// Mitsubishi GX Works2 project: 250627_단일공정순차제어(2)   PLC: Q02U

PROGRAM MAIN
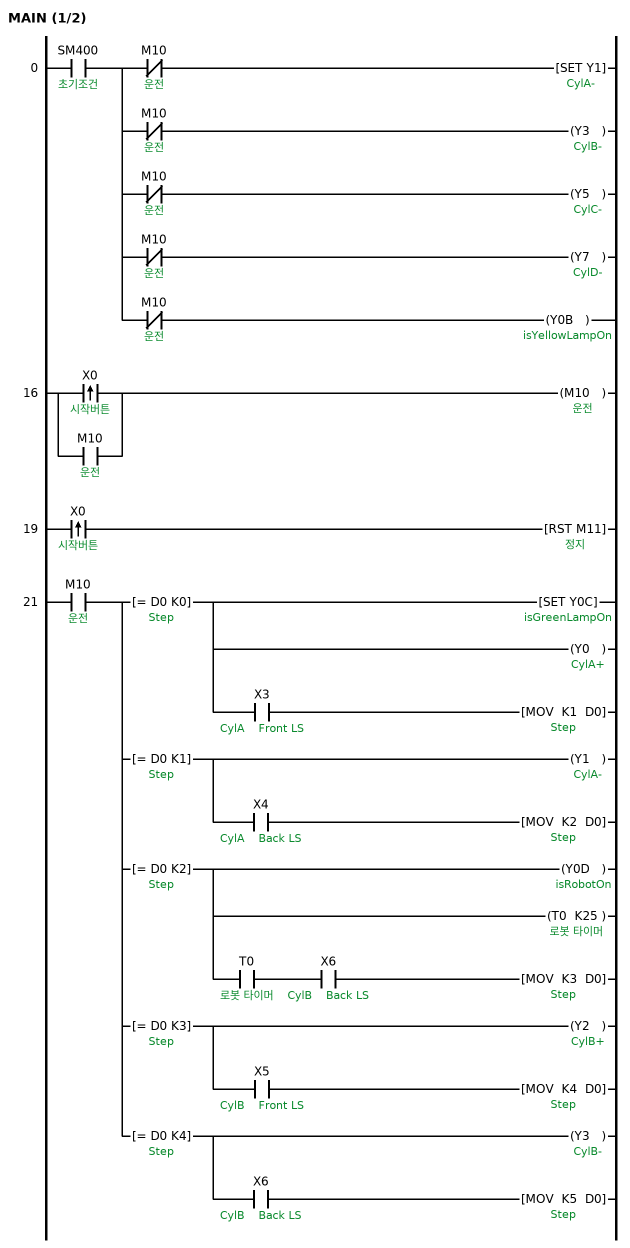
0     LD      SM400  ; 초기조건
      MPS
      ANI     M10  ; 운전
      SET     Y1  ; CylA-
      MRD
      ANI     M10  ; 운전
      OUT     Y3  ; CylB-
      MRD
      ANI     M10  ; 운전
      OUT     Y5  ; CylC-
      MRD
      ANI     M10  ; 운전
      OUT     Y7  ; CylD-
      MPP
      ANI     M10  ; 운전
      OUT     Y0B  ; isYellowLampOn
16    LDP     X0  ; 시작버튼
      OR      M10  ; 운전
      OUT     M10  ; 운전
19    LDP     X0  ; 시작버튼
      RST     M11  ; 정지
21    LD      M10  ; 운전
      MPS
      AND=    D0 K0  ; Step
      SET     Y0C  ; isGreenLampOn
      OUT     Y0  ; CylA+
      AND     X3  ; CylA    Front LS
      MOV     K1 D0
      MRD
      AND=    D0 K1  ; Step
      OUT     Y1  ; CylA-
      AND     X4  ; CylA    Back LS
      MOV     K2 D0
      MRD
      AND=    D0 K2  ; Step
      OUT     Y0D  ; isRobotOn
      OUT     T0 K25  ; 로봇 타이머
      AND     T0  ; 로봇 타이머
      AND     X6  ; CylB    Back LS
      MOV     K3 D0
      MRD
      AND=    D0 K3  ; Step
      OUT     Y2  ; CylB+
      AND     X5  ; CylB    Front LS
      MOV     K4 D0
      MPP
      AND=    D0 K4  ; Step
      OUT     Y3  ; CylB-
      AND     X6  ; CylB    Back LS
      MOV     K5 D0
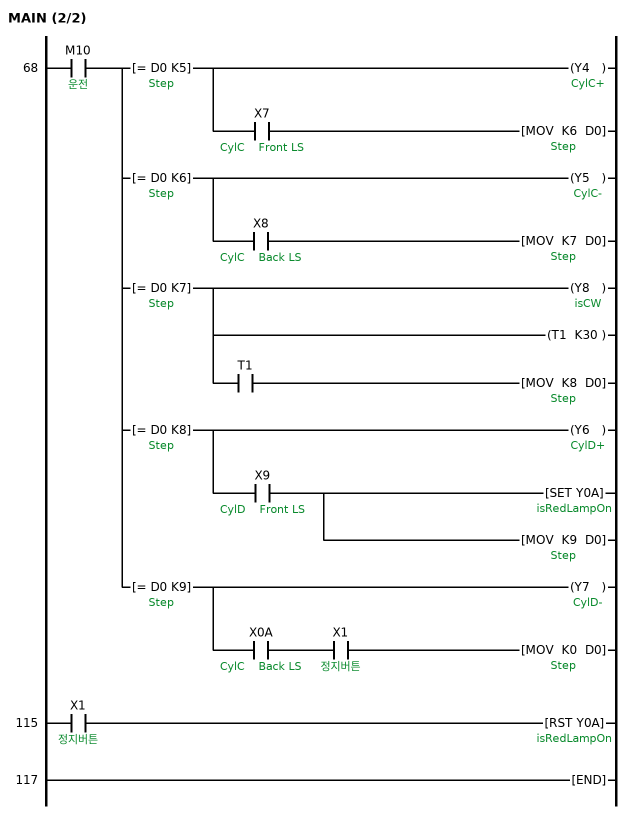
68    LD      M10  ; 운전
      MPS
      AND=    D0 K5  ; Step
      OUT     Y4  ; CylC+
      AND     X7  ; CylC    Front LS
      MOV     K6 D0
      MRD
      AND=    D0 K6  ; Step
      OUT     Y5  ; CylC-
      AND     X8  ; CylC    Back LS
      MOV     K7 D0
      MRD
      AND=    D0 K7  ; Step
      OUT     Y8  ; isCW
      OUT     T1 K30
      AND     T1
      MOV     K8 D0
      MRD
      AND=    D0 K8  ; Step
      OUT     Y6  ; CylD+
      AND     X9  ; CylD    Front LS
      SET     Y0A  ; isRedLampOn
      MOV     K9 D0
      MPP
      AND=    D0 K9  ; Step
      OUT     Y7  ; CylD-
      AND     X0A  ; CylC    Back LS
      AND     X1  ; 정지버튼
      MOV     K0 D0
115   LD      X1  ; 정지버튼
      RST     Y0A  ; isRedLampOn
117   END
END_PROGRAM

// device comments not shown above
X2  ; 긴급정지버튼
X0B  ; CylD    Front LS
X0C  ; CylD    Back LS
X19  ; 근접센서ON
X1A  ; 금속센서ON
Y9  ; isCCW
